// TIA Portal project "GetError_ID_ ve_GetError Locally" (V18)

(* hardware
DEVICE "S7-1200 station_1"  S7-1200 Station
   slot 0: "Rack_0"  S7-1200 Rack  Rack  V1.0
   slot 1: "PLC_1"  CPU 1214C DC/DC/DC  6ES7 214-1AG40-0XB0  V4.6
*)

// ===== PLC "PLC_1"  CPU 1214C DC/DC/DC =====

VAR_GLOBAL   // PLC tag table "Default tag table"
   "Tag_1" AT %I0.0 : Bool;
   "Tag_2" AT %MW10 : Word;
   "Tag_3" AT %Q0.0 : Bool;
END_VAR

DATA_BLOCK "Hata Verileri"   // DB1
{ S7_Optimized_Access := 'TRUE' }
VERSION : 0.1
   VAR
      HATA : ErrorStruct;
   END_VAR
BEGIN
END_DATA_BLOCK

ORGANIZATION_BLOCK "Main"   // OB1, LAD, ProgramCycle
TITLE = "Main Program Sweep (Cycle)"
{ S7_Optimized_Access := 'TRUE' }
VERSION : 0.1
// GetErr_Id komutu çıkışındaki numara hatanın nereden kaynaklandığını gösterir. Programdan kaynaklanan hatayı gösterir. 
// GetErr komutu işletim sistemini çalışma esnasında kaynaklanan hataları gösterir
   VAR_INPUT
      Initial_Call : Bool;   // Initial call of this OB
      Remanence : Bool;   // =True, if remanent data are available
   END_VAR
BEGIN

REGION Network 1
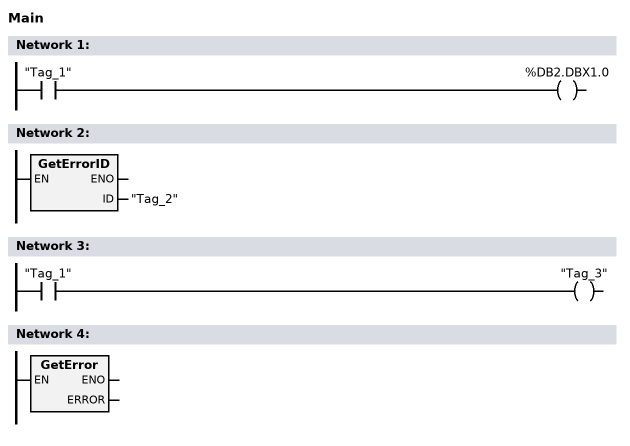
   RUNG wire#powerrail
      Contact( "Tag_1" )
      Coil( %DB2.DBX1.0 )
   END_RUNG
   // the same network as SCL:
   %DB2.DBX1.0 := "Tag_1";
END_REGION

REGION Network 2
   // no SCL statement known for GetErrorID: written as a call
   GetErrorID(id => "Tag_2");
END_REGION

REGION Network 3
   RUNG wire#powerrail
      Contact( "Tag_1" )
      Coil( "Tag_3" )
   END_RUNG
   // the same network as SCL:
   "Tag_3" := "Tag_1";
END_REGION

REGION Network 4
   // no SCL statement known for GetError: written as a call
   GetError();
END_REGION
END_ORGANIZATION_BLOCK